// TIA Portal V20 export
DATA_BLOCK "InstEmDataHmi"   // DB44
TITLE = Instanz von FB EnergyMeterDataToHmi / Instance of FB instance of FB EnergyMeterDataToHmi
AUTHOR : SICAR
FAMILY : Energy
VERSION : 1.0
// Energy meter HMI
// stored: InstanceOfName LSicar_EnMeterDataToHmi, InstanceOfType FB
"LSicar_EnMeterDataToHmi"
   // VAR_INPUT
   //    energyMeter01Visu { ExternalAccessible := 'False'; ExternalVisible := 'False'; ExternalWritable := 'False'} : "LSicar_typeEnMeterVisuStruct";
   //    energyMeter02Visu { ExternalAccessible := 'False'; ExternalVisible := 'False'; ExternalWritable := 'False'} : "LSicar_typeEnMeterVisuStruct";
   //    energyMeter03Visu { ExternalAccessible := 'False'; ExternalVisible := 'False'; ExternalWritable := 'False'} : "LSicar_typeEnMeterVisuStruct";
   //    energyMeter04Visu { ExternalAccessible := 'False'; ExternalVisible := 'False'; ExternalWritable := 'False'} : "LSicar_typeEnMeterVisuStruct";
   //    energyMeter05Visu { ExternalAccessible := 'False'; ExternalVisible := 'False'; ExternalWritable := 'False'} : "LSicar_typeEnMeterVisuStruct";
   //    energyMeter06Visu { ExternalAccessible := 'False'; ExternalVisible := 'False'; ExternalWritable := 'False'} : "LSicar_typeEnMeterVisuStruct";
   //    energyMeter07Visu { ExternalAccessible := 'False'; ExternalVisible := 'False'; ExternalWritable := 'False'} : "LSicar_typeEnMeterVisuStruct";
   //    energyMeter08Visu { ExternalAccessible := 'False'; ExternalVisible := 'False'; ExternalWritable := 'False'} : "LSicar_typeEnMeterVisuStruct";
   // END_VAR
   // VAR
   //    statEmIndex : Int := 1;
   //    statEmData : "LSicar_typeEnMeterVisuStruct";
   //    statResetMinMaxAll : Bool := FALSE;
   //    statResetMinMax : Array[0..8] of Bool;
   //    statResetEnCounterAll : Bool := FALSE;
   //    statResetEnCounter : Array[0..8] of Bool;
   // END_VAR
BEGIN
   energyMeter01Visu.uL1L2 := 480.6464;
   energyMeter01Visu.uL2L3 := 479.3329;
   energyMeter01Visu.uL3L1 := 482.4024;
   energyMeter01Visu.uL1 := 277.0244;
   energyMeter01Visu.uL2 := 283.0648;
   energyMeter01Visu.uL3 := 272.9026;
   energyMeter01Visu.uL1L2Min := 470.1363;
   energyMeter01Visu.uL2L3Min := 469.0945;
   energyMeter01Visu.uL3L1Min := 472.4617;
   energyMeter01Visu.uL1Min := 271.5103;
   energyMeter01Visu.uL2Min := 277.1332;
   energyMeter01Visu.uL3Min := 267.6445;
   energyMeter01Visu.uL1L2Max := 486.0269;
   energyMeter01Visu.uL2L3Max := 484.8441;
   energyMeter01Visu.uL3L1Max := 487.8807;
   energyMeter01Visu.uL1Max := 280.1993;
   energyMeter01Visu.uL2Max := 286.2231;
   energyMeter01Visu.uL3Max := 276.0547;
   energyMeter01Visu.uPhPhAverage := 480.7939;
   energyMeter01Visu.uPhNaverage := 277.6639;
   energyMeter01Visu.uPhPhAverageMin := 470.5642;
   energyMeter01Visu.uPhNaverageMin := 272.105;
   energyMeter01Visu.uPhPhAverageMax := 486.2456;
   energyMeter01Visu.uPhNaverageMax := 280.8176;
   energyMeter01Visu.iL1 := 0.6297245;
   energyMeter01Visu.iL2 := 0.4116209;
   energyMeter01Visu.iL3 := 0.4021624;
   energyMeter01Visu.iL1Min := 0.5503862;
   energyMeter01Visu.iL2Min := 0.3512777;
   energyMeter01Visu.iL3Min := 0.3410119;
   energyMeter01Visu.iL1Max := 2.701323;
   energyMeter01Visu.iL2Max := 2.376321;
   energyMeter01Visu.iL3Max := 1.768756;
   energyMeter01Visu.iAverage := 0.4811693;
   energyMeter01Visu.iAverageMin := 0.4219982;
   energyMeter01Visu.iAverageMax := 2.194234;
   energyMeter01Visu.f := 59.99327;
   energyMeter01Visu.fMin := 59.9567;
   energyMeter01Visu.fMax := 60.07609;
   energyMeter01Visu.sTotal := 400.7156;
   energyMeter01Visu.sTotalMin := 349.7767;
   energyMeter01Visu.sTotalMax := 1823.43;
   energyMeter01Visu.pTotal := 277.3849;
   energyMeter01Visu.pTotalMin := 220.7085;
   energyMeter01Visu.pTotalMax := 670.0833;
   energyMeter01Visu.qTotal := -19.24654;
   energyMeter01Visu.qTotalMin := -422.0206;
   energyMeter01Visu.qTotalMax := -5.418034;
   energyMeter01Visu.cosL1 := 0.8610036;
   energyMeter01Visu.cosL1Min := 0.3576268;
   energyMeter01Visu.cosL1Max := 0.9157406;
   energyMeter01Visu.cosL2 := 0.5061908;
   energyMeter01Visu.cosL2Min := 0.05827232;
   energyMeter01Visu.cosL2Max := 0.7094496;
   energyMeter01Visu.cosL3 := 0.6214478;
   energyMeter01Visu.cosL3Min := 0.1665398;
   energyMeter01Visu.cosL3Max := 0.7301649;
   energyMeter01Visu.cosAverage := 0.6922238;
   energyMeter01Visu.cosAverageMin := 0.2474333;
   energyMeter01Visu.cosAverageMax := 0.7716895;
   energyMeter01Visu.sL1 := 174.449;
   energyMeter01Visu.sL2 := 116.5154;
   energyMeter01Visu.sL3 := 109.7511;
   energyMeter01Visu.sL1Min := 151.7066;
   energyMeter01Visu.sL2Min := 99.03358;
   energyMeter01Visu.sL3Min := 92.7289;
   energyMeter01Visu.sL1Max := 744.3881;
   energyMeter01Visu.sL2Max := 669.9091;
   energyMeter01Visu.sL3Max := 480.3434;
   energyMeter01Visu.pL1 := 150.2012;
   energyMeter01Visu.pL2 := 58.97903;
   energyMeter01Visu.pL3 := 68.20461;
   energyMeter01Visu.pL1Min := 127.6866;
   energyMeter01Visu.pL2Min := 20.87;
   energyMeter01Visu.pL3Min := 52.5906;
   energyMeter01Visu.pL1Max := 281.8818;
   energyMeter01Visu.pL2Max := 194.1828;
   energyMeter01Visu.pL3Max := 220.8245;
   energyMeter01Visu.qL1 := -4.041785;
   energyMeter01Visu.qL2 := 41.25737;
   energyMeter01Visu.qL3 := -56.46213;
   energyMeter01Visu.qL1Min := -144.4171;
   energyMeter01Visu.qL2Min := -98.00859;
   energyMeter01Visu.qL3Min := -198.8008;
   energyMeter01Visu.qL1Max := 28.71266;
   energyMeter01Visu.qL2Max := 50.3845;
   energyMeter01Visu.qL3Max := -53.43742;
   energyMeter01Visu.eActiveRate1Import := 736796.1;
   energyMeter01Visu.eActiveRate2Import := 0.0;
   energyMeter01Visu.eActiveRate1Export := 0.0002530577;
   energyMeter01Visu.eActiveRate2Export := 0.0;
   energyMeter01Visu.eReactiveRate1Import := 5676.457;
   energyMeter01Visu.eReactiveRate2Import := 0.0;
   energyMeter01Visu.eReactiveRate1Export := 293593.3;
   energyMeter01Visu.eReactiveRate2Export := 0.0;
   energyMeter01Visu.eApparentRate1Import := 1470773.0;
   energyMeter01Visu.eApparentRate2Import := 0.0;
   energyMeter01Visu.rTimeDataEnergy := DTL#1970-01-01-00:00:00;
   energyMeter01Visu.rTimeDataValue := DTL#1970-01-01-00:00:00;
   energyMeter01Visu.uPhPhMod := 16#0000;
   energyMeter01Visu.uPhNmod := 16#0000;
   energyMeter01Visu.iMod := 16#0000;
   energyMeter01Visu.sMod := 16#0000;
   energyMeter01Visu.pMod := 16#0000;
   energyMeter01Visu.qMod := 16#0000;
   energyMeter01Visu.eMod := 16#0000;
   energyMeter01Visu.fMod := 16#0000;
   energyMeter01Visu.cosMod := 16#0000;
   energyMeter01Visu.calculateValue1 := 16#0000;
   energyMeter01Visu.calculateValue2 := 16#0000;
   energyMeter01Visu.calculateValue3 := 16#0000;
   energyMeter01Visu.calculateValue4 := 16#0000;
   energyMeter01Visu.calculateValue5 := 16#0000;
   energyMeter01Visu.calculateValue6 := 16#0000;
   energyMeter01Visu.energyMeterUnit := 16#0000;
   energyMeter01Visu.restStartAuto := FALSE;
   energyMeter01Visu.readValue := FALSE;
   energyMeter01Visu.connectionType := 0;
   energyMeter01Visu.driverError := 0;
   energyMeter02Visu.uL1L2 := 0.0;
   energyMeter02Visu.uL2L3 := 0.0;
   energyMeter02Visu.uL3L1 := 0.0;
   energyMeter02Visu.uL1 := 0.0;
   energyMeter02Visu.uL2 := 0.0;
   energyMeter02Visu.uL3 := 0.0;
   energyMeter02Visu.uL1L2Min := 0.0;
   energyMeter02Visu.uL2L3Min := 0.0;
   energyMeter02Visu.uL3L1Min := 0.0;
   energyMeter02Visu.uL1Min := 0.0;
   energyMeter02Visu.uL2Min := 0.0;
   energyMeter02Visu.uL3Min := 0.0;
   energyMeter02Visu.uL1L2Max := 0.0;
   energyMeter02Visu.uL2L3Max := 0.0;
   energyMeter02Visu.uL3L1Max := 0.0;
   energyMeter02Visu.uL1Max := 0.0;
   energyMeter02Visu.uL2Max := 0.0;
   energyMeter02Visu.uL3Max := 0.0;
   energyMeter02Visu.uPhPhAverage := 0.0;
   energyMeter02Visu.uPhNaverage := 0.0;
   energyMeter02Visu.uPhPhAverageMin := 0.0;
   energyMeter02Visu.uPhNaverageMin := 0.0;
   energyMeter02Visu.uPhPhAverageMax := 0.0;
   energyMeter02Visu.uPhNaverageMax := 0.0;
   energyMeter02Visu.iL1 := 0.0;
   energyMeter02Visu.iL2 := 0.0;
   energyMeter02Visu.iL3 := 0.0;
   energyMeter02Visu.iL1Min := 0.0;
   energyMeter02Visu.iL2Min := 0.0;
   energyMeter02Visu.iL3Min := 0.0;
   energyMeter02Visu.iL1Max := 0.0;
   energyMeter02Visu.iL2Max := 0.0;
   energyMeter02Visu.iL3Max := 0.0;
   energyMeter02Visu.iAverage := 0.0;
   energyMeter02Visu.iAverageMin := 0.0;
   energyMeter02Visu.iAverageMax := 0.0;
   energyMeter02Visu.f := 0.0;
   energyMeter02Visu.fMin := 0.0;
   energyMeter02Visu.fMax := 0.0;
   energyMeter02Visu.sTotal := 0.0;
   energyMeter02Visu.sTotalMin := 0.0;
   energyMeter02Visu.sTotalMax := 0.0;
   energyMeter02Visu.pTotal := 0.0;
   energyMeter02Visu.pTotalMin := 0.0;
   energyMeter02Visu.pTotalMax := 0.0;
   energyMeter02Visu.qTotal := 0.0;
   energyMeter02Visu.qTotalMin := 0.0;
   energyMeter02Visu.qTotalMax := 0.0;
   energyMeter02Visu.cosL1 := 0.0;
   energyMeter02Visu.cosL1Min := 0.0;
   energyMeter02Visu.cosL1Max := 0.0;
   energyMeter02Visu.cosL2 := 0.0;
   energyMeter02Visu.cosL2Min := 0.0;
   energyMeter02Visu.cosL2Max := 0.0;
   energyMeter02Visu.cosL3 := 0.0;
   energyMeter02Visu.cosL3Min := 0.0;
   energyMeter02Visu.cosL3Max := 0.0;
   energyMeter02Visu.cosAverage := 0.0;
   energyMeter02Visu.cosAverageMin := 0.0;
   energyMeter02Visu.cosAverageMax := 0.0;
   energyMeter02Visu.sL1 := 0.0;
   energyMeter02Visu.sL2 := 0.0;
   energyMeter02Visu.sL3 := 0.0;
   energyMeter02Visu.sL1Min := 0.0;
   energyMeter02Visu.sL2Min := 0.0;
   energyMeter02Visu.sL3Min := 0.0;
   energyMeter02Visu.sL1Max := 0.0;
   energyMeter02Visu.sL2Max := 0.0;
   energyMeter02Visu.sL3Max := 0.0;
   energyMeter02Visu.pL1 := 0.0;
   energyMeter02Visu.pL2 := 0.0;
   energyMeter02Visu.pL3 := 0.0;
   energyMeter02Visu.pL1Min := 0.0;
   energyMeter02Visu.pL2Min := 0.0;
   energyMeter02Visu.pL3Min := 0.0;
   energyMeter02Visu.pL1Max := 0.0;
   energyMeter02Visu.pL2Max := 0.0;
   energyMeter02Visu.pL3Max := 0.0;
   energyMeter02Visu.qL1 := 0.0;
   energyMeter02Visu.qL2 := 0.0;
   energyMeter02Visu.qL3 := 0.0;
   energyMeter02Visu.qL1Min := 0.0;
   energyMeter02Visu.qL2Min := 0.0;
   energyMeter02Visu.qL3Min := 0.0;
   energyMeter02Visu.qL1Max := 0.0;
   energyMeter02Visu.qL2Max := 0.0;
   energyMeter02Visu.qL3Max := 0.0;
   energyMeter02Visu.eActiveRate1Import := 0.0;
   energyMeter02Visu.eActiveRate2Import := 0.0;
   energyMeter02Visu.eActiveRate1Export := 0.0;
   energyMeter02Visu.eActiveRate2Export := 0.0;
   energyMeter02Visu.eReactiveRate1Import := 0.0;
   energyMeter02Visu.eReactiveRate2Import := 0.0;
   energyMeter02Visu.eReactiveRate1Export := 0.0;
   energyMeter02Visu.eReactiveRate2Export := 0.0;
   energyMeter02Visu.eApparentRate1Import := 0.0;
   energyMeter02Visu.eApparentRate2Import := 0.0;
   energyMeter02Visu.rTimeDataEnergy := DTL#1970-01-01-00:00:00;
   energyMeter02Visu.rTimeDataValue := DTL#1970-01-01-00:00:00;
   energyMeter02Visu.uPhPhMod := 16#0000;
   energyMeter02Visu.uPhNmod := 16#0000;
   energyMeter02Visu.iMod := 16#0000;
   energyMeter02Visu.sMod := 16#0000;
   energyMeter02Visu.pMod := 16#0000;
   energyMeter02Visu.qMod := 16#0000;
   energyMeter02Visu.eMod := 16#0000;
   energyMeter02Visu.fMod := 16#0000;
   energyMeter02Visu.cosMod := 16#0000;
   energyMeter02Visu.calculateValue1 := 16#0000;
   energyMeter02Visu.calculateValue2 := 16#0000;
   energyMeter02Visu.calculateValue3 := 16#0000;
   energyMeter02Visu.calculateValue4 := 16#0000;
   energyMeter02Visu.calculateValue5 := 16#0000;
   energyMeter02Visu.calculateValue6 := 16#0000;
   energyMeter02Visu.energyMeterUnit := 16#0000;
   energyMeter02Visu.restStartAuto := FALSE;
   energyMeter02Visu.readValue := FALSE;
   energyMeter02Visu.connectionType := 0;
   energyMeter02Visu.driverError := 0;
   energyMeter03Visu.uL1L2 := 0.0;
   energyMeter03Visu.uL2L3 := 0.0;
   energyMeter03Visu.uL3L1 := 0.0;
   energyMeter03Visu.uL1 := 0.0;
   energyMeter03Visu.uL2 := 0.0;
   energyMeter03Visu.uL3 := 0.0;
   energyMeter03Visu.uL1L2Min := 0.0;
   energyMeter03Visu.uL2L3Min := 0.0;
   energyMeter03Visu.uL3L1Min := 0.0;
   energyMeter03Visu.uL1Min := 0.0;
   energyMeter03Visu.uL2Min := 0.0;
   energyMeter03Visu.uL3Min := 0.0;
   energyMeter03Visu.uL1L2Max := 0.0;
   energyMeter03Visu.uL2L3Max := 0.0;
   energyMeter03Visu.uL3L1Max := 0.0;
   energyMeter03Visu.uL1Max := 0.0;
   energyMeter03Visu.uL2Max := 0.0;
   energyMeter03Visu.uL3Max := 0.0;
   energyMeter03Visu.uPhPhAverage := 0.0;
   energyMeter03Visu.uPhNaverage := 0.0;
   energyMeter03Visu.uPhPhAverageMin := 0.0;
   energyMeter03Visu.uPhNaverageMin := 0.0;
   energyMeter03Visu.uPhPhAverageMax := 0.0;
   energyMeter03Visu.uPhNaverageMax := 0.0;
   energyMeter03Visu.iL1 := 0.0;
   energyMeter03Visu.iL2 := 0.0;
   energyMeter03Visu.iL3 := 0.0;
   energyMeter03Visu.iL1Min := 0.0;
   energyMeter03Visu.iL2Min := 0.0;
   energyMeter03Visu.iL3Min := 0.0;
   energyMeter03Visu.iL1Max := 0.0;
   energyMeter03Visu.iL2Max := 0.0;
   energyMeter03Visu.iL3Max := 0.0;
   energyMeter03Visu.iAverage := 0.0;
   energyMeter03Visu.iAverageMin := 0.0;
   energyMeter03Visu.iAverageMax := 0.0;
   energyMeter03Visu.f := 0.0;
   energyMeter03Visu.fMin := 0.0;
   energyMeter03Visu.fMax := 0.0;
   energyMeter03Visu.sTotal := 0.0;
   energyMeter03Visu.sTotalMin := 0.0;
   energyMeter03Visu.sTotalMax := 0.0;
   energyMeter03Visu.pTotal := 0.0;
   energyMeter03Visu.pTotalMin := 0.0;
   energyMeter03Visu.pTotalMax := 0.0;
   energyMeter03Visu.qTotal := 0.0;
   energyMeter03Visu.qTotalMin := 0.0;
   energyMeter03Visu.qTotalMax := 0.0;
   energyMeter03Visu.cosL1 := 0.0;
   energyMeter03Visu.cosL1Min := 0.0;
   energyMeter03Visu.cosL1Max := 0.0;
   energyMeter03Visu.cosL2 := 0.0;
   energyMeter03Visu.cosL2Min := 0.0;
   energyMeter03Visu.cosL2Max := 0.0;
   energyMeter03Visu.cosL3 := 0.0;
   energyMeter03Visu.cosL3Min := 0.0;
   energyMeter03Visu.cosL3Max := 0.0;
   energyMeter03Visu.cosAverage := 0.0;
   energyMeter03Visu.cosAverageMin := 0.0;
   energyMeter03Visu.cosAverageMax := 0.0;
   energyMeter03Visu.sL1 := 0.0;
   energyMeter03Visu.sL2 := 0.0;
   energyMeter03Visu.sL3 := 0.0;
   energyMeter03Visu.sL1Min := 0.0;
   energyMeter03Visu.sL2Min := 0.0;
   energyMeter03Visu.sL3Min := 0.0;
   energyMeter03Visu.sL1Max := 0.0;
   energyMeter03Visu.sL2Max := 0.0;
   energyMeter03Visu.sL3Max := 0.0;
   energyMeter03Visu.pL1 := 0.0;
   energyMeter03Visu.pL2 := 0.0;
   energyMeter03Visu.pL3 := 0.0;
   energyMeter03Visu.pL1Min := 0.0;
   energyMeter03Visu.pL2Min := 0.0;
   energyMeter03Visu.pL3Min := 0.0;
   energyMeter03Visu.pL1Max := 0.0;
   energyMeter03Visu.pL2Max := 0.0;
   energyMeter03Visu.pL3Max := 0.0;
   energyMeter03Visu.qL1 := 0.0;
   energyMeter03Visu.qL2 := 0.0;
   energyMeter03Visu.qL3 := 0.0;
   energyMeter03Visu.qL1Min := 0.0;
   energyMeter03Visu.qL2Min := 0.0;
   energyMeter03Visu.qL3Min := 0.0;
   energyMeter03Visu.qL1Max := 0.0;
   energyMeter03Visu.qL2Max := 0.0;
   energyMeter03Visu.qL3Max := 0.0;
   energyMeter03Visu.eActiveRate1Import := 0.0;
   energyMeter03Visu.eActiveRate2Import := 0.0;
   energyMeter03Visu.eActiveRate1Export := 0.0;
   energyMeter03Visu.eActiveRate2Export := 0.0;
   energyMeter03Visu.eReactiveRate1Import := 0.0;
   energyMeter03Visu.eReactiveRate2Import := 0.0;
   energyMeter03Visu.eReactiveRate1Export := 0.0;
   energyMeter03Visu.eReactiveRate2Export := 0.0;
   energyMeter03Visu.eApparentRate1Import := 0.0;
   energyMeter03Visu.eApparentRate2Import := 0.0;
   energyMeter03Visu.rTimeDataEnergy := DTL#1970-01-01-00:00:00;
   energyMeter03Visu.rTimeDataValue := DTL#1970-01-01-00:00:00;
   energyMeter03Visu.uPhPhMod := 16#0000;
   energyMeter03Visu.uPhNmod := 16#0000;
   energyMeter03Visu.iMod := 16#0000;
   energyMeter03Visu.sMod := 16#0000;
   energyMeter03Visu.pMod := 16#0000;
   energyMeter03Visu.qMod := 16#0000;
   energyMeter03Visu.eMod := 16#0000;
   energyMeter03Visu.fMod := 16#0000;
   energyMeter03Visu.cosMod := 16#0000;
   energyMeter03Visu.calculateValue1 := 16#0000;
   energyMeter03Visu.calculateValue2 := 16#0000;
   energyMeter03Visu.calculateValue3 := 16#0000;
   energyMeter03Visu.calculateValue4 := 16#0000;
   energyMeter03Visu.calculateValue5 := 16#0000;
   energyMeter03Visu.calculateValue6 := 16#0000;
   energyMeter03Visu.energyMeterUnit := 16#0000;
   energyMeter03Visu.restStartAuto := FALSE;
   energyMeter03Visu.readValue := FALSE;
   energyMeter03Visu.connectionType := 0;
   energyMeter03Visu.driverError := 0;
   energyMeter04Visu.uL1L2 := 0.0;
   energyMeter04Visu.uL2L3 := 0.0;
   energyMeter04Visu.uL3L1 := 0.0;
   energyMeter04Visu.uL1 := 0.0;
   energyMeter04Visu.uL2 := 0.0;
   energyMeter04Visu.uL3 := 0.0;
   energyMeter04Visu.uL1L2Min := 0.0;
   energyMeter04Visu.uL2L3Min := 0.0;
   energyMeter04Visu.uL3L1Min := 0.0;
   energyMeter04Visu.uL1Min := 0.0;
   energyMeter04Visu.uL2Min := 0.0;
   energyMeter04Visu.uL3Min := 0.0;
   energyMeter04Visu.uL1L2Max := 0.0;
   energyMeter04Visu.uL2L3Max := 0.0;
   energyMeter04Visu.uL3L1Max := 0.0;
   energyMeter04Visu.uL1Max := 0.0;
   energyMeter04Visu.uL2Max := 0.0;
   energyMeter04Visu.uL3Max := 0.0;
   energyMeter04Visu.uPhPhAverage := 0.0;
   energyMeter04Visu.uPhNaverage := 0.0;
   energyMeter04Visu.uPhPhAverageMin := 0.0;
   energyMeter04Visu.uPhNaverageMin := 0.0;
   energyMeter04Visu.uPhPhAverageMax := 0.0;
   energyMeter04Visu.uPhNaverageMax := 0.0;
   energyMeter04Visu.iL1 := 0.0;
   energyMeter04Visu.iL2 := 0.0;
   energyMeter04Visu.iL3 := 0.0;
   energyMeter04Visu.iL1Min := 0.0;
   energyMeter04Visu.iL2Min := 0.0;
   energyMeter04Visu.iL3Min := 0.0;
   energyMeter04Visu.iL1Max := 0.0;
   energyMeter04Visu.iL2Max := 0.0;
   energyMeter04Visu.iL3Max := 0.0;
   energyMeter04Visu.iAverage := 0.0;
   energyMeter04Visu.iAverageMin := 0.0;
   energyMeter04Visu.iAverageMax := 0.0;
   energyMeter04Visu.f := 0.0;
   energyMeter04Visu.fMin := 0.0;
   energyMeter04Visu.fMax := 0.0;
   energyMeter04Visu.sTotal := 0.0;
   energyMeter04Visu.sTotalMin := 0.0;
   energyMeter04Visu.sTotalMax := 0.0;
   energyMeter04Visu.pTotal := 0.0;
   energyMeter04Visu.pTotalMin := 0.0;
   energyMeter04Visu.pTotalMax := 0.0;
   energyMeter04Visu.qTotal := 0.0;
   energyMeter04Visu.qTotalMin := 0.0;
   energyMeter04Visu.qTotalMax := 0.0;
   energyMeter04Visu.cosL1 := 0.0;
   energyMeter04Visu.cosL1Min := 0.0;
   energyMeter04Visu.cosL1Max := 0.0;
   energyMeter04Visu.cosL2 := 0.0;
   energyMeter04Visu.cosL2Min := 0.0;
   energyMeter04Visu.cosL2Max := 0.0;
   energyMeter04Visu.cosL3 := 0.0;
   energyMeter04Visu.cosL3Min := 0.0;
   energyMeter04Visu.cosL3Max := 0.0;
   energyMeter04Visu.cosAverage := 0.0;
   energyMeter04Visu.cosAverageMin := 0.0;
   energyMeter04Visu.cosAverageMax := 0.0;
   energyMeter04Visu.sL1 := 0.0;
   energyMeter04Visu.sL2 := 0.0;
   energyMeter04Visu.sL3 := 0.0;
   energyMeter04Visu.sL1Min := 0.0;
   energyMeter04Visu.sL2Min := 0.0;
   energyMeter04Visu.sL3Min := 0.0;
   energyMeter04Visu.sL1Max := 0.0;
   energyMeter04Visu.sL2Max := 0.0;
   energyMeter04Visu.sL3Max := 0.0;
   energyMeter04Visu.pL1 := 0.0;
   energyMeter04Visu.pL2 := 0.0;
   energyMeter04Visu.pL3 := 0.0;
   energyMeter04Visu.pL1Min := 0.0;
   energyMeter04Visu.pL2Min := 0.0;
   energyMeter04Visu.pL3Min := 0.0;
   energyMeter04Visu.pL1Max := 0.0;
   energyMeter04Visu.pL2Max := 0.0;
   energyMeter04Visu.pL3Max := 0.0;
   energyMeter04Visu.qL1 := 0.0;
   energyMeter04Visu.qL2 := 0.0;
   energyMeter04Visu.qL3 := 0.0;
   energyMeter04Visu.qL1Min := 0.0;
   energyMeter04Visu.qL2Min := 0.0;
   energyMeter04Visu.qL3Min := 0.0;
   energyMeter04Visu.qL1Max := 0.0;
   energyMeter04Visu.qL2Max := 0.0;
   energyMeter04Visu.qL3Max := 0.0;
   energyMeter04Visu.eActiveRate1Import := 0.0;
   energyMeter04Visu.eActiveRate2Import := 0.0;
   energyMeter04Visu.eActiveRate1Export := 0.0;
   energyMeter04Visu.eActiveRate2Export := 0.0;
   energyMeter04Visu.eReactiveRate1Import := 0.0;
   energyMeter04Visu.eReactiveRate2Import := 0.0;
   energyMeter04Visu.eReactiveRate1Export := 0.0;
   energyMeter04Visu.eReactiveRate2Export := 0.0;
   energyMeter04Visu.eApparentRate1Import := 0.0;
   energyMeter04Visu.eApparentRate2Import := 0.0;
   energyMeter04Visu.rTimeDataEnergy := DTL#1970-01-01-00:00:00;
   energyMeter04Visu.rTimeDataValue := DTL#1970-01-01-00:00:00;
   energyMeter04Visu.uPhPhMod := 16#0000;
   energyMeter04Visu.uPhNmod := 16#0000;
   energyMeter04Visu.iMod := 16#0000;
   energyMeter04Visu.sMod := 16#0000;
   energyMeter04Visu.pMod := 16#0000;
   energyMeter04Visu.qMod := 16#0000;
   energyMeter04Visu.eMod := 16#0000;
   energyMeter04Visu.fMod := 16#0000;
   energyMeter04Visu.cosMod := 16#0000;
   energyMeter04Visu.calculateValue1 := 16#0000;
   energyMeter04Visu.calculateValue2 := 16#0000;
   energyMeter04Visu.calculateValue3 := 16#0000;
   energyMeter04Visu.calculateValue4 := 16#0000;
   energyMeter04Visu.calculateValue5 := 16#0000;
   energyMeter04Visu.calculateValue6 := 16#0000;
   energyMeter04Visu.energyMeterUnit := 16#0000;
   energyMeter04Visu.restStartAuto := FALSE;
   energyMeter04Visu.readValue := FALSE;
   energyMeter04Visu.connectionType := 0;
   energyMeter04Visu.driverError := 0;
   energyMeter05Visu.uL1L2 := 0.0;
   energyMeter05Visu.uL2L3 := 0.0;
   energyMeter05Visu.uL3L1 := 0.0;
   energyMeter05Visu.uL1 := 0.0;
   energyMeter05Visu.uL2 := 0.0;
   energyMeter05Visu.uL3 := 0.0;
   energyMeter05Visu.uL1L2Min := 0.0;
   energyMeter05Visu.uL2L3Min := 0.0;
   energyMeter05Visu.uL3L1Min := 0.0;
   energyMeter05Visu.uL1Min := 0.0;
   energyMeter05Visu.uL2Min := 0.0;
   energyMeter05Visu.uL3Min := 0.0;
   energyMeter05Visu.uL1L2Max := 0.0;
   energyMeter05Visu.uL2L3Max := 0.0;
   energyMeter05Visu.uL3L1Max := 0.0;
   energyMeter05Visu.uL1Max := 0.0;
   energyMeter05Visu.uL2Max := 0.0;
   energyMeter05Visu.uL3Max := 0.0;
   energyMeter05Visu.uPhPhAverage := 0.0;
   energyMeter05Visu.uPhNaverage := 0.0;
   energyMeter05Visu.uPhPhAverageMin := 0.0;
   energyMeter05Visu.uPhNaverageMin := 0.0;
   energyMeter05Visu.uPhPhAverageMax := 0.0;
   energyMeter05Visu.uPhNaverageMax := 0.0;
   energyMeter05Visu.iL1 := 0.0;
   energyMeter05Visu.iL2 := 0.0;
   energyMeter05Visu.iL3 := 0.0;
   energyMeter05Visu.iL1Min := 0.0;
   energyMeter05Visu.iL2Min := 0.0;
   energyMeter05Visu.iL3Min := 0.0;
   energyMeter05Visu.iL1Max := 0.0;
   energyMeter05Visu.iL2Max := 0.0;
   energyMeter05Visu.iL3Max := 0.0;
   energyMeter05Visu.iAverage := 0.0;
   energyMeter05Visu.iAverageMin := 0.0;
   energyMeter05Visu.iAverageMax := 0.0;
   energyMeter05Visu.f := 0.0;
   energyMeter05Visu.fMin := 0.0;
   energyMeter05Visu.fMax := 0.0;
   energyMeter05Visu.sTotal := 0.0;
   energyMeter05Visu.sTotalMin := 0.0;
   energyMeter05Visu.sTotalMax := 0.0;
   energyMeter05Visu.pTotal := 0.0;
   energyMeter05Visu.pTotalMin := 0.0;
   energyMeter05Visu.pTotalMax := 0.0;
   energyMeter05Visu.qTotal := 0.0;
   energyMeter05Visu.qTotalMin := 0.0;
   energyMeter05Visu.qTotalMax := 0.0;
   energyMeter05Visu.cosL1 := 0.0;
   energyMeter05Visu.cosL1Min := 0.0;
   energyMeter05Visu.cosL1Max := 0.0;
   energyMeter05Visu.cosL2 := 0.0;
   energyMeter05Visu.cosL2Min := 0.0;
   energyMeter05Visu.cosL2Max := 0.0;
   energyMeter05Visu.cosL3 := 0.0;
   energyMeter05Visu.cosL3Min := 0.0;
   energyMeter05Visu.cosL3Max := 0.0;
   energyMeter05Visu.cosAverage := 0.0;
   energyMeter05Visu.cosAverageMin := 0.0;
   energyMeter05Visu.cosAverageMax := 0.0;
   energyMeter05Visu.sL1 := 0.0;
   energyMeter05Visu.sL2 := 0.0;
   energyMeter05Visu.sL3 := 0.0;
   energyMeter05Visu.sL1Min := 0.0;
   energyMeter05Visu.sL2Min := 0.0;
   energyMeter05Visu.sL3Min := 0.0;
   energyMeter05Visu.sL1Max := 0.0;
   energyMeter05Visu.sL2Max := 0.0;
   energyMeter05Visu.sL3Max := 0.0;
   energyMeter05Visu.pL1 := 0.0;
   energyMeter05Visu.pL2 := 0.0;
   energyMeter05Visu.pL3 := 0.0;
   energyMeter05Visu.pL1Min := 0.0;
   energyMeter05Visu.pL2Min := 0.0;
   energyMeter05Visu.pL3Min := 0.0;
   energyMeter05Visu.pL1Max := 0.0;
   energyMeter05Visu.pL2Max := 0.0;
   energyMeter05Visu.pL3Max := 0.0;
   energyMeter05Visu.qL1 := 0.0;
   energyMeter05Visu.qL2 := 0.0;
   energyMeter05Visu.qL3 := 0.0;
   energyMeter05Visu.qL1Min := 0.0;
   energyMeter05Visu.qL2Min := 0.0;
   energyMeter05Visu.qL3Min := 0.0;
   energyMeter05Visu.qL1Max := 0.0;
   energyMeter05Visu.qL2Max := 0.0;
   energyMeter05Visu.qL3Max := 0.0;
   energyMeter05Visu.eActiveRate1Import := 0.0;
   energyMeter05Visu.eActiveRate2Import := 0.0;
   energyMeter05Visu.eActiveRate1Export := 0.0;
   energyMeter05Visu.eActiveRate2Export := 0.0;
   energyMeter05Visu.eReactiveRate1Import := 0.0;
   energyMeter05Visu.eReactiveRate2Import := 0.0;
   energyMeter05Visu.eReactiveRate1Export := 0.0;
   energyMeter05Visu.eReactiveRate2Export := 0.0;
   energyMeter05Visu.eApparentRate1Import := 0.0;
   energyMeter05Visu.eApparentRate2Import := 0.0;
   energyMeter05Visu.rTimeDataEnergy := DTL#1970-01-01-00:00:00;
   energyMeter05Visu.rTimeDataValue := DTL#1970-01-01-00:00:00;
   energyMeter05Visu.uPhPhMod := 16#0000;
   energyMeter05Visu.uPhNmod := 16#0000;
   energyMeter05Visu.iMod := 16#0000;
   energyMeter05Visu.sMod := 16#0000;
   energyMeter05Visu.pMod := 16#0000;
   energyMeter05Visu.qMod := 16#0000;
   energyMeter05Visu.eMod := 16#0000;
   energyMeter05Visu.fMod := 16#0000;
   energyMeter05Visu.cosMod := 16#0000;
   energyMeter05Visu.calculateValue1 := 16#0000;
   energyMeter05Visu.calculateValue2 := 16#0000;
   energyMeter05Visu.calculateValue3 := 16#0000;
   energyMeter05Visu.calculateValue4 := 16#0000;
   energyMeter05Visu.calculateValue5 := 16#0000;
   energyMeter05Visu.calculateValue6 := 16#0000;
   energyMeter05Visu.energyMeterUnit := 16#0000;
   energyMeter05Visu.restStartAuto := FALSE;
   energyMeter05Visu.readValue := FALSE;
   energyMeter05Visu.connectionType := 0;
   energyMeter05Visu.driverError := 0;
   energyMeter06Visu.uL1L2 := 0.0;
   energyMeter06Visu.uL2L3 := 0.0;
   energyMeter06Visu.uL3L1 := 0.0;
   energyMeter06Visu.uL1 := 0.0;
   energyMeter06Visu.uL2 := 0.0;
   energyMeter06Visu.uL3 := 0.0;
   energyMeter06Visu.uL1L2Min := 0.0;
   energyMeter06Visu.uL2L3Min := 0.0;
   energyMeter06Visu.uL3L1Min := 0.0;
   energyMeter06Visu.uL1Min := 0.0;
   energyMeter06Visu.uL2Min := 0.0;
   energyMeter06Visu.uL3Min := 0.0;
   energyMeter06Visu.uL1L2Max := 0.0;
   energyMeter06Visu.uL2L3Max := 0.0;
   energyMeter06Visu.uL3L1Max := 0.0;
   energyMeter06Visu.uL1Max := 0.0;
   energyMeter06Visu.uL2Max := 0.0;
   energyMeter06Visu.uL3Max := 0.0;
   energyMeter06Visu.uPhPhAverage := 0.0;
   energyMeter06Visu.uPhNaverage := 0.0;
   energyMeter06Visu.uPhPhAverageMin := 0.0;
   energyMeter06Visu.uPhNaverageMin := 0.0;
   energyMeter06Visu.uPhPhAverageMax := 0.0;
   energyMeter06Visu.uPhNaverageMax := 0.0;
   energyMeter06Visu.iL1 := 0.0;
   energyMeter06Visu.iL2 := 0.0;
   energyMeter06Visu.iL3 := 0.0;
   energyMeter06Visu.iL1Min := 0.0;
   energyMeter06Visu.iL2Min := 0.0;
   energyMeter06Visu.iL3Min := 0.0;
   energyMeter06Visu.iL1Max := 0.0;
   energyMeter06Visu.iL2Max := 0.0;
   energyMeter06Visu.iL3Max := 0.0;
   energyMeter06Visu.iAverage := 0.0;
   energyMeter06Visu.iAverageMin := 0.0;
   energyMeter06Visu.iAverageMax := 0.0;
   energyMeter06Visu.f := 0.0;
   energyMeter06Visu.fMin := 0.0;
   energyMeter06Visu.fMax := 0.0;
   energyMeter06Visu.sTotal := 0.0;
   energyMeter06Visu.sTotalMin := 0.0;
   energyMeter06Visu.sTotalMax := 0.0;
   energyMeter06Visu.pTotal := 0.0;
   energyMeter06Visu.pTotalMin := 0.0;
   energyMeter06Visu.pTotalMax := 0.0;
   energyMeter06Visu.qTotal := 0.0;
   energyMeter06Visu.qTotalMin := 0.0;
   energyMeter06Visu.qTotalMax := 0.0;
   energyMeter06Visu.cosL1 := 0.0;
   energyMeter06Visu.cosL1Min := 0.0;
   energyMeter06Visu.cosL1Max := 0.0;
   energyMeter06Visu.cosL2 := 0.0;
   energyMeter06Visu.cosL2Min := 0.0;
   energyMeter06Visu.cosL2Max := 0.0;
   energyMeter06Visu.cosL3 := 0.0;
   energyMeter06Visu.cosL3Min := 0.0;
   energyMeter06Visu.cosL3Max := 0.0;
   energyMeter06Visu.cosAverage := 0.0;
   energyMeter06Visu.cosAverageMin := 0.0;
   energyMeter06Visu.cosAverageMax := 0.0;
   energyMeter06Visu.sL1 := 0.0;
   energyMeter06Visu.sL2 := 0.0;
   energyMeter06Visu.sL3 := 0.0;
   energyMeter06Visu.sL1Min := 0.0;
   energyMeter06Visu.sL2Min := 0.0;
   energyMeter06Visu.sL3Min := 0.0;
   energyMeter06Visu.sL1Max := 0.0;
   energyMeter06Visu.sL2Max := 0.0;
   energyMeter06Visu.sL3Max := 0.0;
   energyMeter06Visu.pL1 := 0.0;
   energyMeter06Visu.pL2 := 0.0;
   energyMeter06Visu.pL3 := 0.0;
   energyMeter06Visu.pL1Min := 0.0;
   energyMeter06Visu.pL2Min := 0.0;
   energyMeter06Visu.pL3Min := 0.0;
   energyMeter06Visu.pL1Max := 0.0;
   energyMeter06Visu.pL2Max := 0.0;
   energyMeter06Visu.pL3Max := 0.0;
   energyMeter06Visu.qL1 := 0.0;
   energyMeter06Visu.qL2 := 0.0;
   energyMeter06Visu.qL3 := 0.0;
   energyMeter06Visu.qL1Min := 0.0;
   energyMeter06Visu.qL2Min := 0.0;
   energyMeter06Visu.qL3Min := 0.0;
   energyMeter06Visu.qL1Max := 0.0;
   energyMeter06Visu.qL2Max := 0.0;
   energyMeter06Visu.qL3Max := 0.0;
   energyMeter06Visu.eActiveRate1Import := 0.0;
   energyMeter06Visu.eActiveRate2Import := 0.0;
   energyMeter06Visu.eActiveRate1Export := 0.0;
   energyMeter06Visu.eActiveRate2Export := 0.0;
   energyMeter06Visu.eReactiveRate1Import := 0.0;
   energyMeter06Visu.eReactiveRate2Import := 0.0;
   energyMeter06Visu.eReactiveRate1Export := 0.0;
   energyMeter06Visu.eReactiveRate2Export := 0.0;
   energyMeter06Visu.eApparentRate1Import := 0.0;
   energyMeter06Visu.eApparentRate2Import := 0.0;
   energyMeter06Visu.rTimeDataEnergy := DTL#1970-01-01-00:00:00;
   energyMeter06Visu.rTimeDataValue := DTL#1970-01-01-00:00:00;
   energyMeter06Visu.uPhPhMod := 16#0000;
   energyMeter06Visu.uPhNmod := 16#0000;
   energyMeter06Visu.iMod := 16#0000;
   energyMeter06Visu.sMod := 16#0000;
   energyMeter06Visu.pMod := 16#0000;
   energyMeter06Visu.qMod := 16#0000;
   energyMeter06Visu.eMod := 16#0000;
   energyMeter06Visu.fMod := 16#0000;
   energyMeter06Visu.cosMod := 16#0000;
   energyMeter06Visu.calculateValue1 := 16#0000;
   energyMeter06Visu.calculateValue2 := 16#0000;
   energyMeter06Visu.calculateValue3 := 16#0000;
   energyMeter06Visu.calculateValue4 := 16#0000;
   energyMeter06Visu.calculateValue5 := 16#0000;
   energyMeter06Visu.calculateValue6 := 16#0000;
   energyMeter06Visu.energyMeterUnit := 16#0000;
   energyMeter06Visu.restStartAuto := FALSE;
   energyMeter06Visu.readValue := FALSE;
   energyMeter06Visu.connectionType := 0;
   energyMeter06Visu.driverError := 0;
   energyMeter07Visu.uL1L2 := 0.0;
   energyMeter07Visu.uL2L3 := 0.0;
   energyMeter07Visu.uL3L1 := 0.0;
   energyMeter07Visu.uL1 := 0.0;
   energyMeter07Visu.uL2 := 0.0;
   energyMeter07Visu.uL3 := 0.0;
   energyMeter07Visu.uL1L2Min := 0.0;
   energyMeter07Visu.uL2L3Min := 0.0;
   energyMeter07Visu.uL3L1Min := 0.0;
   energyMeter07Visu.uL1Min := 0.0;
   energyMeter07Visu.uL2Min := 0.0;
   energyMeter07Visu.uL3Min := 0.0;
   energyMeter07Visu.uL1L2Max := 0.0;
   energyMeter07Visu.uL2L3Max := 0.0;
   energyMeter07Visu.uL3L1Max := 0.0;
   energyMeter07Visu.uL1Max := 0.0;
   energyMeter07Visu.uL2Max := 0.0;
   energyMeter07Visu.uL3Max := 0.0;
   energyMeter07Visu.uPhPhAverage := 0.0;
   energyMeter07Visu.uPhNaverage := 0.0;
   energyMeter07Visu.uPhPhAverageMin := 0.0;
   energyMeter07Visu.uPhNaverageMin := 0.0;
   energyMeter07Visu.uPhPhAverageMax := 0.0;
   energyMeter07Visu.uPhNaverageMax := 0.0;
   energyMeter07Visu.iL1 := 0.0;
   energyMeter07Visu.iL2 := 0.0;
   energyMeter07Visu.iL3 := 0.0;
   energyMeter07Visu.iL1Min := 0.0;
   energyMeter07Visu.iL2Min := 0.0;
   energyMeter07Visu.iL3Min := 0.0;
   energyMeter07Visu.iL1Max := 0.0;
   energyMeter07Visu.iL2Max := 0.0;
   energyMeter07Visu.iL3Max := 0.0;
   energyMeter07Visu.iAverage := 0.0;
   energyMeter07Visu.iAverageMin := 0.0;
   energyMeter07Visu.iAverageMax := 0.0;
   energyMeter07Visu.f := 0.0;
   energyMeter07Visu.fMin := 0.0;
   energyMeter07Visu.fMax := 0.0;
   energyMeter07Visu.sTotal := 0.0;
   energyMeter07Visu.sTotalMin := 0.0;
   energyMeter07Visu.sTotalMax := 0.0;
   energyMeter07Visu.pTotal := 0.0;
   energyMeter07Visu.pTotalMin := 0.0;
   energyMeter07Visu.pTotalMax := 0.0;
   energyMeter07Visu.qTotal := 0.0;
   energyMeter07Visu.qTotalMin := 0.0;
   energyMeter07Visu.qTotalMax := 0.0;
   energyMeter07Visu.cosL1 := 0.0;
   energyMeter07Visu.cosL1Min := 0.0;
   energyMeter07Visu.cosL1Max := 0.0;
   energyMeter07Visu.cosL2 := 0.0;
   energyMeter07Visu.cosL2Min := 0.0;
   energyMeter07Visu.cosL2Max := 0.0;
   energyMeter07Visu.cosL3 := 0.0;
   energyMeter07Visu.cosL3Min := 0.0;
   energyMeter07Visu.cosL3Max := 0.0;
   energyMeter07Visu.cosAverage := 0.0;
   energyMeter07Visu.cosAverageMin := 0.0;
   energyMeter07Visu.cosAverageMax := 0.0;
   energyMeter07Visu.sL1 := 0.0;
   energyMeter07Visu.sL2 := 0.0;
   energyMeter07Visu.sL3 := 0.0;
   energyMeter07Visu.sL1Min := 0.0;
   energyMeter07Visu.sL2Min := 0.0;
   energyMeter07Visu.sL3Min := 0.0;
   energyMeter07Visu.sL1Max := 0.0;
   energyMeter07Visu.sL2Max := 0.0;
   energyMeter07Visu.sL3Max := 0.0;
   energyMeter07Visu.pL1 := 0.0;
   energyMeter07Visu.pL2 := 0.0;
   energyMeter07Visu.pL3 := 0.0;
   energyMeter07Visu.pL1Min := 0.0;
   energyMeter07Visu.pL2Min := 0.0;
   energyMeter07Visu.pL3Min := 0.0;
   energyMeter07Visu.pL1Max := 0.0;
   energyMeter07Visu.pL2Max := 0.0;
   energyMeter07Visu.pL3Max := 0.0;
   energyMeter07Visu.qL1 := 0.0;
   energyMeter07Visu.qL2 := 0.0;
   energyMeter07Visu.qL3 := 0.0;
   energyMeter07Visu.qL1Min := 0.0;
   energyMeter07Visu.qL2Min := 0.0;
   energyMeter07Visu.qL3Min := 0.0;
   energyMeter07Visu.qL1Max := 0.0;
   energyMeter07Visu.qL2Max := 0.0;
   energyMeter07Visu.qL3Max := 0.0;
   energyMeter07Visu.eActiveRate1Import := 0.0;
   energyMeter07Visu.eActiveRate2Import := 0.0;
   energyMeter07Visu.eActiveRate1Export := 0.0;
   energyMeter07Visu.eActiveRate2Export := 0.0;
   energyMeter07Visu.eReactiveRate1Import := 0.0;
   energyMeter07Visu.eReactiveRate2Import := 0.0;
   energyMeter07Visu.eReactiveRate1Export := 0.0;
   energyMeter07Visu.eReactiveRate2Export := 0.0;
   energyMeter07Visu.eApparentRate1Import := 0.0;
   energyMeter07Visu.eApparentRate2Import := 0.0;
   energyMeter07Visu.rTimeDataEnergy := DTL#1970-01-01-00:00:00;
   energyMeter07Visu.rTimeDataValue := DTL#1970-01-01-00:00:00;
   energyMeter07Visu.uPhPhMod := 16#0000;
   energyMeter07Visu.uPhNmod := 16#0000;
   energyMeter07Visu.iMod := 16#0000;
   energyMeter07Visu.sMod := 16#0000;
   energyMeter07Visu.pMod := 16#0000;
   energyMeter07Visu.qMod := 16#0000;
   energyMeter07Visu.eMod := 16#0000;
   energyMeter07Visu.fMod := 16#0000;
   energyMeter07Visu.cosMod := 16#0000;
   energyMeter07Visu.calculateValue1 := 16#0000;
   energyMeter07Visu.calculateValue2 := 16#0000;
   energyMeter07Visu.calculateValue3 := 16#0000;
   energyMeter07Visu.calculateValue4 := 16#0000;
   energyMeter07Visu.calculateValue5 := 16#0000;
   energyMeter07Visu.calculateValue6 := 16#0000;
   energyMeter07Visu.energyMeterUnit := 16#0000;
   energyMeter07Visu.restStartAuto := FALSE;
   energyMeter07Visu.readValue := FALSE;
   energyMeter07Visu.connectionType := 0;
   energyMeter07Visu.driverError := 0;
   energyMeter08Visu.uL1L2 := 0.0;
   energyMeter08Visu.uL2L3 := 0.0;
   energyMeter08Visu.uL3L1 := 0.0;
   energyMeter08Visu.uL1 := 0.0;
   energyMeter08Visu.uL2 := 0.0;
   energyMeter08Visu.uL3 := 0.0;
   energyMeter08Visu.uL1L2Min := 0.0;
   energyMeter08Visu.uL2L3Min := 0.0;
   energyMeter08Visu.uL3L1Min := 0.0;
   energyMeter08Visu.uL1Min := 0.0;
   energyMeter08Visu.uL2Min := 0.0;
   energyMeter08Visu.uL3Min := 0.0;
   energyMeter08Visu.uL1L2Max := 0.0;
   energyMeter08Visu.uL2L3Max := 0.0;
   energyMeter08Visu.uL3L1Max := 0.0;
   energyMeter08Visu.uL1Max := 0.0;
   energyMeter08Visu.uL2Max := 0.0;
   energyMeter08Visu.uL3Max := 0.0;
   energyMeter08Visu.uPhPhAverage := 0.0;
   energyMeter08Visu.uPhNaverage := 0.0;
   energyMeter08Visu.uPhPhAverageMin := 0.0;
   energyMeter08Visu.uPhNaverageMin := 0.0;
   energyMeter08Visu.uPhPhAverageMax := 0.0;
   energyMeter08Visu.uPhNaverageMax := 0.0;
   energyMeter08Visu.iL1 := 0.0;
   energyMeter08Visu.iL2 := 0.0;
   energyMeter08Visu.iL3 := 0.0;
   energyMeter08Visu.iL1Min := 0.0;
   energyMeter08Visu.iL2Min := 0.0;
   energyMeter08Visu.iL3Min := 0.0;
   energyMeter08Visu.iL1Max := 0.0;
   energyMeter08Visu.iL2Max := 0.0;
   energyMeter08Visu.iL3Max := 0.0;
   energyMeter08Visu.iAverage := 0.0;
   energyMeter08Visu.iAverageMin := 0.0;
   energyMeter08Visu.iAverageMax := 0.0;
   energyMeter08Visu.f := 0.0;
   energyMeter08Visu.fMin := 0.0;
   energyMeter08Visu.fMax := 0.0;
   energyMeter08Visu.sTotal := 0.0;
   energyMeter08Visu.sTotalMin := 0.0;
   energyMeter08Visu.sTotalMax := 0.0;
   energyMeter08Visu.pTotal := 0.0;
   energyMeter08Visu.pTotalMin := 0.0;
   energyMeter08Visu.pTotalMax := 0.0;
   energyMeter08Visu.qTotal := 0.0;
   energyMeter08Visu.qTotalMin := 0.0;
   energyMeter08Visu.qTotalMax := 0.0;
   energyMeter08Visu.cosL1 := 0.0;
   energyMeter08Visu.cosL1Min := 0.0;
   energyMeter08Visu.cosL1Max := 0.0;
   energyMeter08Visu.cosL2 := 0.0;
   energyMeter08Visu.cosL2Min := 0.0;
   energyMeter08Visu.cosL2Max := 0.0;
   energyMeter08Visu.cosL3 := 0.0;
   energyMeter08Visu.cosL3Min := 0.0;
   energyMeter08Visu.cosL3Max := 0.0;
   energyMeter08Visu.cosAverage := 0.0;
   energyMeter08Visu.cosAverageMin := 0.0;
   energyMeter08Visu.cosAverageMax := 0.0;
   energyMeter08Visu.sL1 := 0.0;
   energyMeter08Visu.sL2 := 0.0;
   energyMeter08Visu.sL3 := 0.0;
   energyMeter08Visu.sL1Min := 0.0;
   energyMeter08Visu.sL2Min := 0.0;
   energyMeter08Visu.sL3Min := 0.0;
   energyMeter08Visu.sL1Max := 0.0;
   energyMeter08Visu.sL2Max := 0.0;
   energyMeter08Visu.sL3Max := 0.0;
   energyMeter08Visu.pL1 := 0.0;
   energyMeter08Visu.pL2 := 0.0;
   energyMeter08Visu.pL3 := 0.0;
   energyMeter08Visu.pL1Min := 0.0;
   energyMeter08Visu.pL2Min := 0.0;
   energyMeter08Visu.pL3Min := 0.0;
   energyMeter08Visu.pL1Max := 0.0;
   energyMeter08Visu.pL2Max := 0.0;
   energyMeter08Visu.pL3Max := 0.0;
   energyMeter08Visu.qL1 := 0.0;
   energyMeter08Visu.qL2 := 0.0;
   energyMeter08Visu.qL3 := 0.0;
   energyMeter08Visu.qL1Min := 0.0;
   energyMeter08Visu.qL2Min := 0.0;
   energyMeter08Visu.qL3Min := 0.0;
   energyMeter08Visu.qL1Max := 0.0;
   energyMeter08Visu.qL2Max := 0.0;
   energyMeter08Visu.qL3Max := 0.0;
   energyMeter08Visu.eActiveRate1Import := 0.0;
   energyMeter08Visu.eActiveRate2Import := 0.0;
   energyMeter08Visu.eActiveRate1Export := 0.0;
   energyMeter08Visu.eActiveRate2Export := 0.0;
   energyMeter08Visu.eReactiveRate1Import := 0.0;
   energyMeter08Visu.eReactiveRate2Import := 0.0;
   energyMeter08Visu.eReactiveRate1Export := 0.0;
   energyMeter08Visu.eReactiveRate2Export := 0.0;
   energyMeter08Visu.eApparentRate1Import := 0.0;
   energyMeter08Visu.eApparentRate2Import := 0.0;
   energyMeter08Visu.rTimeDataEnergy := DTL#1970-01-01-00:00:00;
   energyMeter08Visu.rTimeDataValue := DTL#1970-01-01-00:00:00;
   energyMeter08Visu.uPhPhMod := 16#0000;
   energyMeter08Visu.uPhNmod := 16#0000;
   energyMeter08Visu.iMod := 16#0000;
   energyMeter08Visu.sMod := 16#0000;
   energyMeter08Visu.pMod := 16#0000;
   energyMeter08Visu.qMod := 16#0000;
   energyMeter08Visu.eMod := 16#0000;
   energyMeter08Visu.fMod := 16#0000;
   energyMeter08Visu.cosMod := 16#0000;
   energyMeter08Visu.calculateValue1 := 16#0000;
   energyMeter08Visu.calculateValue2 := 16#0000;
   energyMeter08Visu.calculateValue3 := 16#0000;
   energyMeter08Visu.calculateValue4 := 16#0000;
   energyMeter08Visu.calculateValue5 := 16#0000;
   energyMeter08Visu.calculateValue6 := 16#0000;
   energyMeter08Visu.energyMeterUnit := 16#0000;
   energyMeter08Visu.restStartAuto := FALSE;
   energyMeter08Visu.readValue := FALSE;
   energyMeter08Visu.connectionType := 0;
   energyMeter08Visu.driverError := 0;
   statEmData.uL1L2 := 480.6464;
   statEmData.uL2L3 := 479.3329;
   statEmData.uL3L1 := 482.4024;
   statEmData.uL1 := 277.0244;
   statEmData.uL2 := 283.0648;
   statEmData.uL3 := 272.9026;
   statEmData.uL1L2Min := 470.1363;
   statEmData.uL2L3Min := 469.0945;
   statEmData.uL3L1Min := 472.4617;
   statEmData.uL1Min := 271.5103;
   statEmData.uL2Min := 277.1332;
   statEmData.uL3Min := 267.6445;
   statEmData.uL1L2Max := 486.0269;
   statEmData.uL2L3Max := 484.8441;
   statEmData.uL3L1Max := 487.8807;
   statEmData.uL1Max := 280.1993;
   statEmData.uL2Max := 286.2231;
   statEmData.uL3Max := 276.0547;
   statEmData.uPhPhAverage := 480.7939;
   statEmData.uPhNaverage := 277.6639;
   statEmData.uPhPhAverageMin := 470.5642;
   statEmData.uPhNaverageMin := 272.105;
   statEmData.uPhPhAverageMax := 486.2456;
   statEmData.uPhNaverageMax := 280.8176;
   statEmData.iL1 := 0.6297245;
   statEmData.iL2 := 0.4116209;
   statEmData.iL3 := 0.4021624;
   statEmData.iL1Min := 0.5503862;
   statEmData.iL2Min := 0.3512777;
   statEmData.iL3Min := 0.3410119;
   statEmData.iL1Max := 2.701323;
   statEmData.iL2Max := 2.376321;
   statEmData.iL3Max := 1.768756;
   statEmData.iAverage := 0.4811693;
   statEmData.iAverageMin := 0.4219982;
   statEmData.iAverageMax := 2.194234;
   statEmData.f := 59.99327;
   statEmData.fMin := 59.9567;
   statEmData.fMax := 60.07609;
   statEmData.sTotal := 400.7156;
   statEmData.sTotalMin := 349.7767;
   statEmData.sTotalMax := 1823.43;
   statEmData.pTotal := 277.3849;
   statEmData.pTotalMin := 220.7085;
   statEmData.pTotalMax := 670.0833;
   statEmData.qTotal := -19.24654;
   statEmData.qTotalMin := -422.0206;
   statEmData.qTotalMax := -5.418034;
   statEmData.cosL1 := 0.8610036;
   statEmData.cosL1Min := 0.3576268;
   statEmData.cosL1Max := 0.9157406;
   statEmData.cosL2 := 0.5061908;
   statEmData.cosL2Min := 0.05827232;
   statEmData.cosL2Max := 0.7094496;
   statEmData.cosL3 := 0.6214478;
   statEmData.cosL3Min := 0.1665398;
   statEmData.cosL3Max := 0.7301649;
   statEmData.cosAverage := 0.6922238;
   statEmData.cosAverageMin := 0.2474333;
   statEmData.cosAverageMax := 0.7716895;
   statEmData.sL1 := 174.449;
   statEmData.sL2 := 116.5154;
   statEmData.sL3 := 109.7511;
   statEmData.sL1Min := 151.7066;
   statEmData.sL2Min := 99.03358;
   statEmData.sL3Min := 92.7289;
   statEmData.sL1Max := 744.3881;
   statEmData.sL2Max := 669.9091;
   statEmData.sL3Max := 480.3434;
   statEmData.pL1 := 150.2012;
   statEmData.pL2 := 58.97903;
   statEmData.pL3 := 68.20461;
   statEmData.pL1Min := 127.6866;
   statEmData.pL2Min := 20.87;
   statEmData.pL3Min := 52.5906;
   statEmData.pL1Max := 281.8818;
   statEmData.pL2Max := 194.1828;
   statEmData.pL3Max := 220.8245;
   statEmData.qL1 := -4.041785;
   statEmData.qL2 := 41.25737;
   statEmData.qL3 := -56.46213;
   statEmData.qL1Min := -144.4171;
   statEmData.qL2Min := -98.00859;
   statEmData.qL3Min := -198.8008;
   statEmData.qL1Max := 28.71266;
   statEmData.qL2Max := 50.3845;
   statEmData.qL3Max := -53.43742;
   statEmData.eActiveRate1Import := 736796.1;
   statEmData.eActiveRate2Import := 0.0;
   statEmData.eActiveRate1Export := 0.0002530577;
   statEmData.eActiveRate2Export := 0.0;
   statEmData.eReactiveRate1Import := 5676.457;
   statEmData.eReactiveRate2Import := 0.0;
   statEmData.eReactiveRate1Export := 293593.3;
   statEmData.eReactiveRate2Export := 0.0;
   statEmData.eApparentRate1Import := 1470773.0;
   statEmData.eApparentRate2Import := 0.0;
   statEmData.rTimeDataEnergy := DTL#1970-01-01-00:00:00;
   statEmData.rTimeDataValue := DTL#1970-01-01-00:00:00;
   statEmData.uPhPhMod := 16#0000;
   statEmData.uPhNmod := 16#0000;
   statEmData.iMod := 16#0000;
   statEmData.sMod := 16#0000;
   statEmData.pMod := 16#0000;
   statEmData.qMod := 16#0000;
   statEmData.eMod := 16#0000;
   statEmData.fMod := 16#0000;
   statEmData.cosMod := 16#0000;
   statEmData.calculateValue1 := 16#0000;
   statEmData.calculateValue2 := 16#0000;
   statEmData.calculateValue3 := 16#0000;
   statEmData.calculateValue4 := 16#0000;
   statEmData.calculateValue5 := 16#0000;
   statEmData.calculateValue6 := 16#0000;
   statEmData.energyMeterUnit := 16#0000;
   statEmData.restStartAuto := FALSE;
   statEmData.readValue := FALSE;
   statEmData.connectionType := 0;
   statEmData.driverError := 0;
   statResetMinMax[0..8] := FALSE;
   statResetEnCounter[0..8] := FALSE;
END_DATA_BLOCK
